TYPE CMD_RackFeeder :
STRUCT
	cmd			: E_RackFeederCmd;
	nId			: INT;
END_STRUCT
END_TYPE

(* stored: Version 1.1.0.1
   DUT CMD_RackFeeder: Id {3aa38b58-a16f-4499-bc13-e1e11d0feba2} *)
